# EPICS substitutions: evrSupport/Db/bsa/bsaATTREdef2.substitutions
#==============================================================================
#
# Abs:  Beam Synchronous Acquisition records for a single Toroid.
#
# Name: bsaATTREdef.substitutions
#
# Note: Must follow the LCLS naming conventions.
#
#==============================================================================
# BSA Integration Note:
# Each device attribute (such as width ) provides input to bsaEdefAvg.db.
# The bsaEdefAvg.db provides the RMS and Avg -$(DEV):$(SECN)<edef id>, and history -
#   $(DEV):$(SECN)HST<edef id> for each device attribute for each of 20 edefs.
#
file bsaEdefAvg2.db
{
#	      Device   Name                                                      Init
#                                                                                Event Code
  pattern {  DEV ,  SECN , INP ,DESC   ,MD,MDID , EGU  ,HOPR ,LOPR ,PREC ,ADEL ,  NSAM, SIZE             }
	  { $(D) ,$(ATTR), $(I),  1    , 1,  1  ,$(EG) ,$(HO),$(LO),$(PR),$(AD),  2800, $(SINK_SIZE\=10) }
	  { $(D) ,$(ATTR), $(I),  2    , 2,  2  ,$(EG) ,$(HO),$(LO),$(PR),$(AD),  2800, $(SINK_SIZE\=10) }
	  { $(D) ,$(ATTR), $(I),  3    , 3,  3  ,$(EG) ,$(HO),$(LO),$(PR),$(AD),  2800, $(SINK_SIZE\=10) }
	  { $(D) ,$(ATTR), $(I),  4    , 4,  4  ,$(EG) ,$(HO),$(LO),$(PR),$(AD),  2800, $(SINK_SIZE\=10) }
	  { $(D) ,$(ATTR), $(I),  5    , 5,  5  ,$(EG) ,$(HO),$(LO),$(PR),$(AD),  2800, $(SINK_SIZE\=10) }
	  { $(D) ,$(ATTR), $(I),  6    , 6,  6  ,$(EG) ,$(HO),$(LO),$(PR),$(AD),  2800, $(SINK_SIZE\=10) }
	  { $(D) ,$(ATTR), $(I),  7    , 7,  7  ,$(EG) ,$(HO),$(LO),$(PR),$(AD),  2800, $(SINK_SIZE\=10) }
	  { $(D) ,$(ATTR), $(I),  8    , 8,  8  ,$(EG) ,$(HO),$(LO),$(PR),$(AD),  2800, $(SINK_SIZE\=10) }
	  { $(D) ,$(ATTR), $(I),  9    , 9,  9  ,$(EG) ,$(HO),$(LO),$(PR),$(AD),  2800, $(SINK_SIZE\=10) }
	  { $(D) ,$(ATTR), $(I),  10   ,10,  10 ,$(EG) ,$(HO),$(LO),$(PR),$(AD),  2800, $(SINK_SIZE\=10) }
	  { $(D) ,$(ATTR), $(I),  11   ,11,  11 ,$(EG) ,$(HO),$(LO),$(PR),$(AD),  2800, $(SINK_SIZE\=10) }
	  { $(D) ,$(ATTR), $(I),  CUS1H,12,  CUS1H ,$(EG) ,$(HO),$(LO),$(PR),$(AD),  2800, $(SINK_SIZE\=1) }
	  { $(D) ,$(ATTR), $(I),  CUSTH,13,  CUSTH ,$(EG) ,$(HO),$(LO),$(PR),$(AD),  2800, $(SINK_SIZE\=1) }
	  { $(D) ,$(ATTR), $(I),  CUSBR,14,  CUSBR ,$(EG) ,$(HO),$(LO),$(PR),$(AD),  2800, $(SINK_SIZE\=1) }
	  { $(D) ,$(ATTR), $(I),  CUH1H,15,  CUH1H ,$(EG) ,$(HO),$(LO),$(PR),$(AD),  2800, $(SINK_SIZE\=1) }
	  { $(D) ,$(ATTR), $(I),  1H   ,16,  1H    ,$(EG) ,$(HO),$(LO),$(PR),$(AD),  2800, $(SINK_SIZE\=1) }
	  { $(D) ,$(ATTR), $(I),  TH   ,17,  TH    ,$(EG) ,$(HO),$(LO),$(PR),$(AD),  2800, $(SINK_SIZE\=1) }
	  { $(D) ,$(ATTR), $(I),  BR   ,18,  BR    ,$(EG) ,$(HO),$(LO),$(PR),$(AD),  2800, $(SINK_SIZE\=1) }
	  { $(D) ,$(ATTR), $(I),  CUHTH,19,  CUHTH ,$(EG) ,$(HO),$(LO),$(PR),$(AD),  2800, $(SINK_SIZE\=1) }
	  { $(D) ,$(ATTR), $(I),  CUHBR,20,  CUHBR ,$(EG) ,$(HO),$(LO),$(PR),$(AD),  2800, $(SINK_SIZE\=1) }
}
